// Mitsubishi GX Works2 project: practice3   PLC: Q03UDV

PROGRAM MAIN
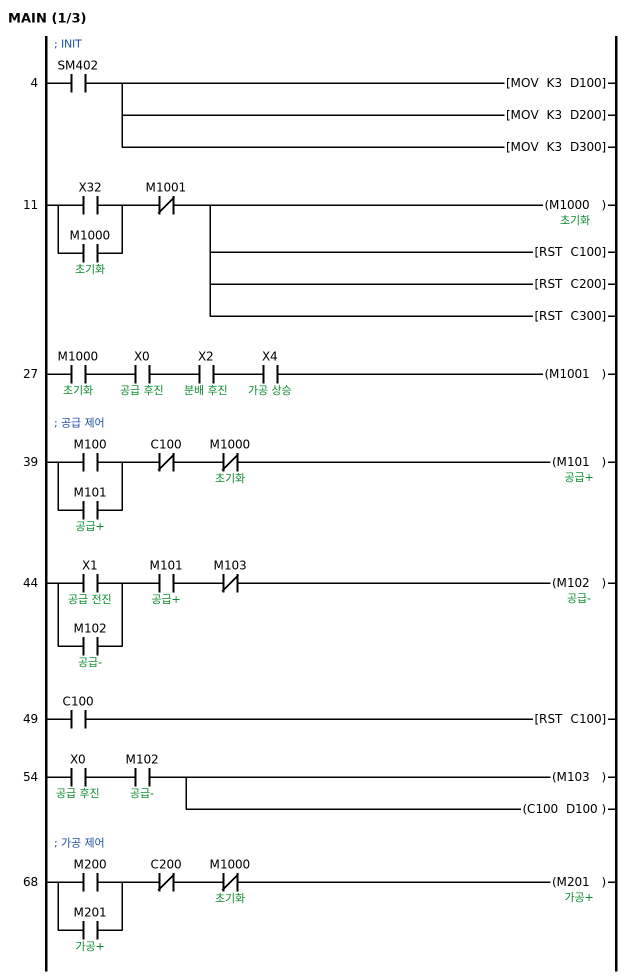
; INIT
4     LD      SM402
      MOV     K3 D100
      MOV     K3 D200
      MOV     K3 D300
11    LD      X32
      OR      M1000  ; 초기화
      ANI     M1001
      OUT     M1000  ; 초기화
      RST     C100
      RST     C200
      RST     C300
27    LD      M1000  ; 초기화
      AND     X0  ; 공급 후진
      AND     X2  ; 분배 후진
      AND     X4  ; 가공 상승
      OUT     M1001
; 공급 제어
39    LD      M100
      OR      M101  ; 공급+
      ANI     C100
      ANI     M1000  ; 초기화
      OUT     M101  ; 공급+
44    LD      X1  ; 공급 전진
      OR      M102  ; 공급-
      AND     M101  ; 공급+
      ANI     M103
      OUT     M102  ; 공급-
49    LD      C100
      RST     C100
54    LD      X0  ; 공급 후진
      AND     M102  ; 공급-
      OUT     M103
      OUT     C100 D100
; 가공 제어
68    LD      M200
      OR      M201  ; 가공+
      ANI     C200
      ANI     M1000  ; 초기화
      OUT     M201  ; 가공+
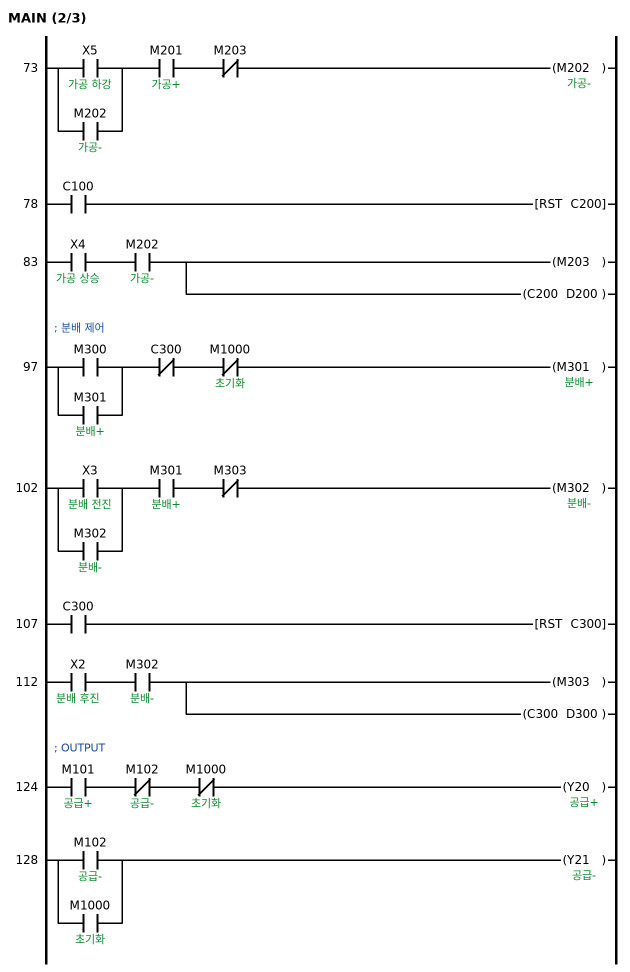
73    LD      X5  ; 가공 하강
      OR      M202  ; 가공-
      AND     M201  ; 가공+
      ANI     M203
      OUT     M202  ; 가공-
78    LD      C100
      RST     C200
83    LD      X4  ; 가공 상승
      AND     M202  ; 가공-
      OUT     M203
      OUT     C200 D200
; 분배 제어
97    LD      M300
      OR      M301  ; 분배+
      ANI     C300
      ANI     M1000  ; 초기화
      OUT     M301  ; 분배+
102   LD      X3  ; 분배 전진
      OR      M302  ; 분배-
      AND     M301  ; 분배+
      ANI     M303
      OUT     M302  ; 분배-
107   LD      C300
      RST     C300
112   LD      X2  ; 분배 후진
      AND     M302  ; 분배-
      OUT     M303
      OUT     C300 D300
; OUTPUT
124   LD      M101  ; 공급+
      ANI     M102  ; 공급-
      ANI     M1000  ; 초기화
      OUT     Y20  ; 공급+
128   LD      M102  ; 공급-
      OR      M1000  ; 초기화
      OUT     Y21  ; 공급-
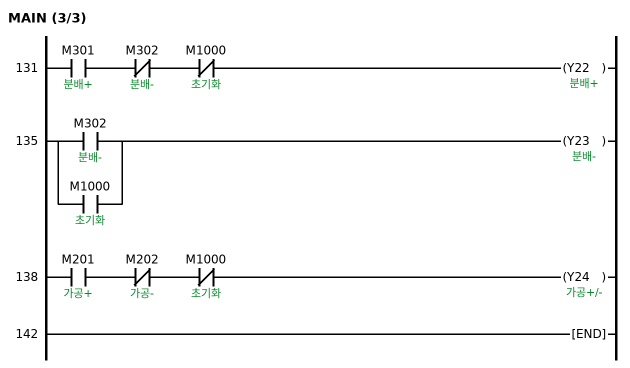
131   LD      M301  ; 분배+
      ANI     M302  ; 분배-
      ANI     M1000  ; 초기화
      OUT     Y22  ; 분배+
135   LD      M302  ; 분배-
      OR      M1000  ; 초기화
      OUT     Y23  ; 분배-
138   LD      M201  ; 가공+
      ANI     M202  ; 가공-
      ANI     M1000  ; 초기화
      OUT     Y24  ; 가공+/-
142   END
END_PROGRAM

// device comments not shown above
M10  ; 공급 동작
M11  ; 분배 동작
M12  ; 가공 동작
